// Mitsubishi GX Works2 project: alarmManager   PLC: FX3G
// Базовая структура управления вентиляциооной установкой

// global labels: Global1
VAR_GLOBAL
  xSeason AT M11 : BOOL;
  dO_PumpStart AT M10 : BOOL;
  aO_1 AT D10 : REAL;
  aO_2 AT D11 : REAL;
  xAlarm AT M1 : BOOL;
  xUserStart AT M0 : BOOL;
  AI_Temp AT D500 : INT;
  DI_KM1 AT X000 : BOOL;
  DO_Motor AT Y000 : BOOL;
  xCriticalAlarm AT M2 : BOOL;
  alarmReset AT M3 : BOOL;
  statusAlarm AT M4 : BOOL;
  statusCritical AT M5 : BOOL;
END_VAR

// task Task_01 (event TRUE, interval 0, priority 31): POU_01
// task Init (event M8002, interval 0, priority 24): Init
// task Process (event FALSE, interval T#150ms, priority 29): Process
// user libraries (not included): alarmManager

PROGRAM Init
VAR
  aInit : A_init;
END_VAR
(*Init Alarms *)
	AL_D_START := 3000; (* Start alarms library*)
	AL_NUMS := 32; (*Numbers of events *)
	
	(* Critical Alarm signals*)

	(*  fbAmInit(iNum := 3, iSeverity :=4, iProcess :=1, xLock := TRUE, xLatch := TRUE,  xBuzzer := TRUE ); *)  (*Freeze alarm *)
	aInit(iNum:= 0 ,iSeverity:= 2 ,iProcess:= 1 ,xLatch:= FALSE,xBuzzer:= TRUE , xLock:= TRUE);
	aInit(iNum:= 1 ,iSeverity:= 3 ,iProcess:= 2 ,xLatch:= TRUE ,xBuzzer:= TRUE , xLock:= TRUE );

	 


(* *)
END_PROGRAM

PROGRAM POU_01
VAR
  iStep : INT;
  xInit : BOOL;
END_VAR
(* RST( MEP( xManualWorks ) , xAutoWorks );
RST( MEP(xAutoWorks ) ,xManualWorks  );  *)
(* System can work only in one state Auto or Manual There is constol change*)

 		IF xInit = 0 THEN  iStep := 0 ; 
 		ELSE 
 			iStep := 10;
 		END_IF; (* Проверяем была ли выполнена инициализация xInit = 1 Ули была то переходим на шаг 10 если нет - на шаг 0 *)

CASE iStep OF
	0: (* Init  - Инициализация Задаем начальные значения переменным*)
	IF xInit = 0  THEN 

			IF xSeason =1 THEN
					dO_PumpStart := 1;
				ELSE 
					dO_PumpStart := 0;
			END_IF; 
			IF MEP(xAlarm) THEN (*Проверка на наличие ошибок Если есть то переходим на шаг 100 для их отработки *)
					iStep := 100;
				ELSE
					xInit := 1;
					aO_1 := 0.0;
					aO_2 := 0.0;
					iStep := 10;
			END_IF;
	END_IF;

	
	10: (* Base *)
	

	
	IF xUserStart = 1 THEN 
		iStep := 20;
		ELSE 
		iStep := 10;
	END_IF;

	100: (* Alarm *)
		;
	END_CASE;



(*	
D500 := D100Z1;

IF MEP( M8013) AND xUserStart = TRUE  THEN
	icountMin := icountMin +1;
	IF icountMin =8 THEN
		icountMin := 0;

	END_IF;
END_IF; 
*)
END_PROGRAM

PROGRAM Process
VAR
  alSet : A_set;
  varSET : BOOL;
  alReset : A_reset;
  alStatus : A_status;
END_VAR
	(* aSet(EN:= varSET,iNum:= 1 , xState:= xSeason , ENO:=  xAlarm ); *)
alSet(iNum:= 0, xState:= xSeason, Q := xCriticalAlarm);
alSet(iNum:= 1, xState:= xSeason, Q := xAlarm );

alReset(reset:= alarmReset );
alStatus(ALARM:= statusAlarm ,CRITICAL:= statusCritical );

(* BON( varSET, D0Z4 , 1 , xAlarm ); *)

(*Freeze Alarm *)
;
(* *)

(* *)

(* *)
;
(* *)
END_PROGRAM

FUNCTION SeasonControl
VAR_INPUT
  tempOut : INT;  (* Temp Outdore - Температура наружнего воздуха *)
  tempWinter : INT;  (* Temp for switch on Winter - Уставка перехода на Зимний режим *)
  tempSummer : INT;  (* Temp for switch on Summer - Уставка перехода на летний режим *)
  triger : BOOL;  (* 1 - was switch to winter 0 - was switch to summer *)
END_VAR
IF tempOut  <  tempWinter THEN 
		SeasonControl := 1; (* Output  Set flag - 1  to force switching to Winter *)
	ELSE 
		IF tempOut  > tempSummer THEN 
			SeasonControl := 0; (* Output  Set flag - 0  to force switching to Summer*)
		ELSE 
			SeasonControl := triger; (* Don't change r*)
		END_IF;

	END_IF;
END_FUNCTION

FUNCTION TestFunction
TestFunction := TRUE;
END_FUNCTION
